ABB RobotStudio station: Tp2_20201216-022622.rsstn

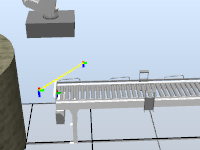
Station Tp2 (saved by RobotStudio 20.2.9116.0)
Controller Controlador1
  mechanical unit ROB_1: IRB660_180_315__01_2, 6 joints, base frame (0, 0, 1500) mm
Layout (positions relative to the parent item):
  - transporteCajas [part, from Equipment\Conveyor Guide 400.rslib] at (0, 1500, 0) mm, rotated rx 0 ry 0 rz 90 deg
  - Euro Pallet [graphiccomponentgroup, from Equipment\Euro Pallet.rslib] at (1000, -1425, 435) mm
    - Body 1 [part, from Equipment\Euro Pallet.rslib]
  - transportePallets [part, from Equipment\Conveyor 950 4000 h2.rslib] at (1000, -1500, 0) mm
  - IRB660_180_315__01_2 [mechanism, from Robots\IRB660_180_315__01.rslib] at (0, 0, 1500) mm; joint values [1.7033, 0.3901, 1.218, 1.7033] (rad or m)
  - ventosa_tool [mechanism] at (-200, 1500, 1970) mm, rotated rx 180 ry 0 rz 180 deg
      TCP ventosa_tool at (0, 0, 200) mm
      links: ventosa
  - fuenteBloques [smart component] at (-200, 1500, 770) mm
      signals: DI agarrar, DO cajaLista
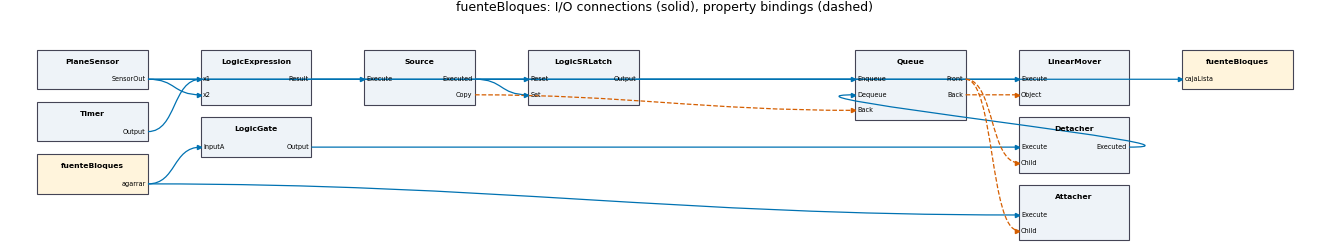
      connections:
        LogicSRLatch.Output -> LinearMover.Execute
        PlaneSensor.SensorOut -> LogicSRLatch.Reset
        Timer.Output -> LogicExpression.x1
        PlaneSensor.SensorOut -> LogicExpression.x2
        LogicExpression.Result -> Source.Execute
        Source.Executed -> LogicSRLatch.Set
        PlaneSensor.SensorOut -> fuenteBloques.cajaLista
        fuenteBloques.agarrar -> Attacher.Execute
        LogicGate.Output -> Detacher.Execute
        fuenteBloques.agarrar -> LogicGate.InputA
        Source.Executed -> Queue.Enqueue
        Detacher.Executed -> Queue.Dequeue
        Source.Copy => Queue.Back
        Queue.Front => Attacher.Child
        Queue.Front => Detacher.Child
        Queue.Back => LinearMover.Object
    - Source [smart component, from Components\Source.rslib]
        properties: Source=caja; Copy=(none); Parent=(none); Position=[0 2.5 0]; Orientation=[0 0 0]; Transient=true; PhysicsBehavior=0
    - Timer [smart component, from Components\Timer.rslib]
        properties: StartTime=0; Interval=5; Repeat=true; CurrentTime=106.92
    - LinearMover [smart component, from Components\LinearMover.rslib]
        properties: Object=(none); Direction=[0 2.5 0]; Speed=-0.8; Reference=Local; ReferenceObject=fuenteBloques
    - PlaneSensor [smart component, from Components\PlaneSensor.rslib]
        properties: Origin=[-0.1 0.00100000000000011 0]; Axis1=[0 0 0.2]; Axis2=[0.2 0 0]; SensedPart=(none)
      - _sensorPart_ [part]
    - Queue [smart component, from Components\Queue.rslib]
        properties: Back=(none); Front=(none); Queue={173b848c-cad7-4bfa-9db7-b362a6be6541};{42a1e277-da34-4a99-8a7e-8b7e8b7e7cc9};{04dbb89d-5868-4f29-bd88-e772b263fe2b};{3bc43ee5-764c-4884-9fd4-1b708219fe3c};{af3e8c9d-81ed-4749-abec-f1d859ddef08};{e6c2343c-3b22-41cc-a537-5f9a15884bd1};{c5bca7ae-cffb-460c-8184-5ba0c64709a5};{747dc2ab-9ebc-4d75-8dd9-eb3637d21ba6}; NumberOfObjects=1
    - caja [part]
    - LogicSRLatch [smart component, from Components\LogicSRLatch.rslib]
    - LogicExpression [smart component, from Components\LogicExpression.rslib]
        properties: Expression=x1 AND NOT x2
    - Attacher [smart component, from Components\Attacher.rslib]
        properties: Parent=ventosa_tool; Flange=0; Child=(none); Mount=false; Offset=[0 0 0]; Orientation=[0 0 0]
    - Detacher [smart component, from Components\Detacher.rslib]
        properties: Child=(none); KeepPosition=true
    - StopSimulation [smart component, from Components\StopSimulation.rslib]
    - StopSimulation_2 [smart component, from Components\StopSimulation.rslib]
    - LogicGate [smart component, from Components\LogicGate.rslib]
        properties: Operator=NOT; Delay=0
  - Pieza_1 [part]
Attachment: Euro Pallet is attached to transportePallets
Attachment: ventosa_tool is attached to IRB660_180_315__01_2 / Link6
Attachment: pistaCajas is attached to transporteCajas
Attachment: pistaPallets is attached to transportePallets
Station logic (signal -> signal, property => property):
  Controlador1.do_pick -> fuenteBloques.agarrar
  fuenteBloques.cajaLista -> Controlador1.cajaLista
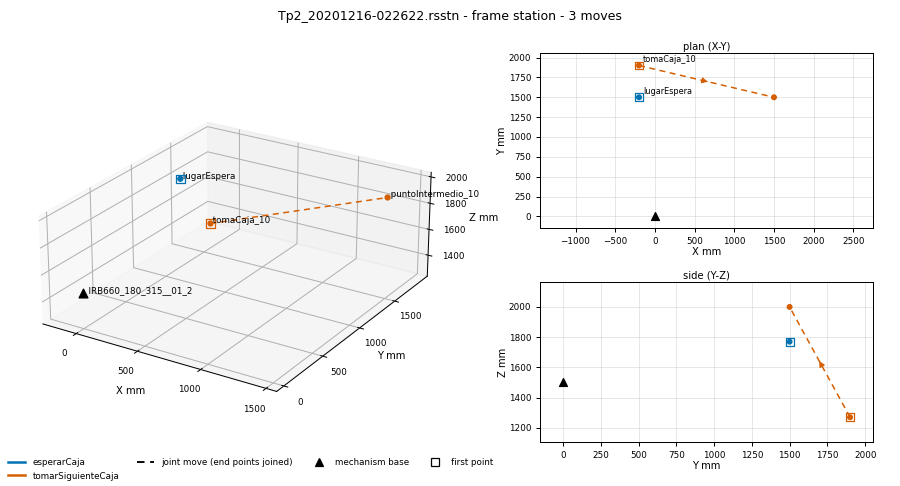
[picture p0: tool path of Tp2_20201216-022622.rsstn in frame station, 3 of 3 moves have a stored position in this frame; points joined in program order, loops and branches not executed]
Targets, tools, work objects and paths stored in the station, written as RAPID:
! task T_ROB1
MODULE Module1
  PERS tooldata ventosa_tool:=[TRUE,[[0,0,200],[1,0,0,0]],[1,[0,0,1],[1,0,0,0],0,0,0]];
  PERS wobjdata pistaCajas:=[FALSE,TRUE,"",[[-200,1500,770],[0,0,1,0]],[[0,0,0],[1,0,0,0]]];
  PERS wobjdata pistaPallets:=[FALSE,TRUE,"",[[1000,-1425,579],[0,0,1,0]],[[0,0,0],[1,0,0,0]]];
  CONST robtarget lugarEspera:=[[0,0,-1000],[1,0,0,0],[0,0,0,0],[9E+09,9E+09,9E+09,9E+09,9E+09,9E+09]];
  CONST robtarget tomaCaja_10:=[[0,400,-500],[1,0,0,0],[0,0,0,0],[9E+09,9E+09,9E+09,9E+09,9E+09,9E+09]];
  CONST robtarget superficiePallet_10:=[[0,0,0],[1,0,0,0],[0,0,0,0],[9E+09,9E+09,9E+09,9E+09,9E+09,9E+09]];
  CONST robtarget puntoIntermedio_10:=[[1500,1500,2000],[0,0,1,0],[0,0,0,0],[9E+09,9E+09,9E+09,9E+09,9E+09,9E+09]];
  PROC main()
    SetDO do_pick,0;
    esperarCaja;
    tomarSiguienteCaja;
    esperarCaja;
  ENDPROC
  PROC esperarCaja()
    MoveJ lugarEspera,v1000,fine,ventosa_tool\WObj:=pistaCajas;
    WaitDI cajaLista,1;
  ENDPROC
  PROC tomarSiguienteCaja()
    MoveJ tomaCaja_10,v1000,fine,ventosa_tool\WObj:=pistaCajas;
    SetDO do_pick,1;
    WaitTime 0.2;
    MoveJ puntoIntermedio_10,v1000,z100,ventosa_tool\WObj:=wobj0;
  ENDPROC
ENDMODULE

